TYPE ST_WorkOrder :
STRUCT
	IDWorkOrder		: LINT; (* Identificatore univoco dell'ordine di lavoro *)
	State			: INT; (* Stato dell'ordine di lavoro : 1=DA ESEGUIRE,2=IN ESECUZIONE,3=TERMINATO *)
	Support			: ST_SupportData; (* Struttura descrizione supporto *)
	Layer 			: ST_LayerData; (* Struttura descrizione falda *)
	SlabNumber  	: INT; (* Numero di lastre da depositare sul supporto *)
	SlabDimension 	: ST_DimensionElement; (* Dimensione Lastra *)
	LayerSequence 	: INT; (* Sequenza di deposito delle falde -> 0=Nessuna falda,1=Deposito dopo ogni lastra,2=Deposito ogni 2 lastre,ecc*)
	ReadyToChange	: INT; (* Se = 1, la macchina è pronta a eseguire il cambio ordine *) 
END_STRUCT
END_TYPE

(* stored: Version 1.1.0.1, ProductVersion 3.1.4024.11
   DUT ST_WorkOrder: Id {c2f3def5-3177-41ce-be7d-09f0cef80ce4} *)
